FUNCTION_BLOCK RadioBool (* Composite Function Block Type *)
  (* Standard: 61499-2 *)
  (* Version 0.0, 15/08/2022, Pranay Jhunjhunwala, Schneider Electric, template *)
  PACKAGE Main;
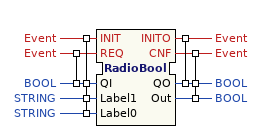
  EVENT_INPUT
    INIT WITH QI, Label1, Label0; (* Initialization Request *)
    REQ WITH QI; (* Normal Execution Request *)
  END_EVENT
  EVENT_OUTPUT
    INITO WITH QO; (* Initialization Confirm *)
    CNF WITH QO, Out; (* Execution Confirmation *)
  END_EVENT
  VAR_INPUT
    QI : BOOL; (* Input event qualifier *)
    Label1 : STRING;
    Label0 : STRING;
  END_VAR
  VAR_OUTPUT
    QO : BOOL; (* Output event qualifier *)
    Out : BOOL;
  END_VAR
  FBS
    IThis : RadioBool_HMI;
  END_FBS
  EVENT_CONNECTIONS
    INIT TO IThis.INIT;
    REQ TO IThis.REQ;
    IThis.INITO TO INITO;
    IThis.CNF TO CNF;
    IThis.INITO TO IThis.REQ;
  END_CONNECTIONS
  DATA_CONNECTIONS
    QI TO IThis.QI;
    Label1 TO IThis.Label1;
    Label0 TO IThis.Label0;
    IThis.Out TO Out;
    IThis.QO TO QO;
  END_CONNECTIONS
END_FUNCTION_BLOCK
